RESOURCE_TYPE top
  (* Standard: 61499-2 *)
  (* Version 0.1, 2017-00-25, hpea485, UOA *)
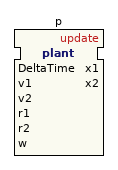
  FBS
    p : plant;
  END_FBS
END_RESOURCE_TYPE
